TYPE ST_SeedLiftSys :
STRUCT
END_STRUCT
END_TYPE

(* stored: Version 1.1.0.1, ProductVersion 3.1.4024.12
   DUT ST_SeedLiftSys: Id {31ce2740-e6f1-48fe-a015-7700d2a24f0e} *)
